# B&R Automation Studio project Stojan2
Automation Studio 4.0.18.71 SP

## Configuration Config1

CPU , AutomationRuntime P3.09, Build 4.1.2

### Task classes (Cpu.sw)
```

```

### Hardware
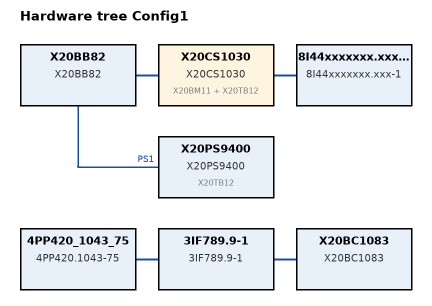
```
3IF789.9-1 : 3IF789.9-1 v1.1.3.0  [SS -> 4PP420_1043_75.SS1]
4PP420_1043_75 : 4PP420.1043-75 v1.0.0.0
  Cyclic1Duration = 10000
  Cyclic1Tolerance = 10000
  Cyclic2Duration = 20000
  Cyclic2Tolerance = 20000
  Cyclic3Duration = 50000
  Cyclic3Tolerance = 50000
  Cyclic4Duration = 100000
  Cyclic4Tolerance = 100000
  Cyclic5Duration = 200000
  Cyclic5Tolerance = 200000
  Cyclic6Duration = 500000
  Cyclic6Tolerance = 500000
  Cyclic7Duration = 1000000
  Cyclic7Tolerance = 1000000
  Cyclic8Duration = 10000
  Cyclic8Tolerance = 30000000
8I44xxxxxxx.xxx-1 : 8I44xxxxxxx.xxx-1 v1.1.3.0  [SER1 -> X20CS1030.IF1 (NodeNumber=10)]
  Supervision = off
  COD = 0
X20BB82 : X20BB82 v1.0.0.0
  Connector IF1:
    CycleTime = 1000
X20BC1083 : X20BC1083 v1.3.6.0  [PLK1 -> 3IF789.9-1.IF2 (NodeNumber=1); SL -> X20BB82.SL1]
X20BM11 : X20BM11 v1.0.0.0  [X2X1 -> X20BB82.IF1]
X20CS1030 : X20CS1030 v1.3.0.0  [SS1 -> X20TB12a.SS; SL -> X20BM11.SL1]
  Connector IF1:
    Baudrate = 19200
    DeviceType = RS485
    ActivateMODBUSRTU = 1
X20PS9400 : X20PS9400 v1.0.2.0  [SS1 -> X20TB12.SS; PS -> X20BB82.PS1]
X20TB12 : X20TB12 v1.0.0.0
X20TB12a : X20TB12 v1.0.0.0
```

## Logical view

Binary libraries used (declarations not repeated): operator, runtime, astime, AsIecCon, AsIOAcc


### Program Logical/ACPi (IEC)

#### ACPi.st - Cyclic code
```iecst
(********************************************************************
 * COPYRIGHT --
 ********************************************************************
 * Program: ACPi
 * File: ACPi.st
 * Author: vancurar
 * Created: 22.10.2012
 ********************************************************************
 * Implementation of program ACPi
 ********************************************************************)

PROGRAM _INIT
	LFRD_Output;

END_PROGRAM

PROGRAM _CYCLIC

	CASE ETAD_Input AND 16#FF  OF
		16#40, 16#50: (* Switch on disabled *)
		CMDD_Output := 16#0006;

		16#21, 16#31: (*Ready to switch on *)
		IF switchOn THEN
			CMDD_Output := 16#0007;
		END_IF

		16#33, 16#23: (*Switched on *)
		CMDD_Output := 16#000F;

		16#37, 16#27: (*Operation enabled *)
		IF NOT switchOn THEN
			CMDD_Output := 16#0006;
		END_IF

		IF quickStop THEN
			CMDD_Output := 16#0002;
		END_IF

		16#17, 16#07: (*Quick stop active *)
		quickStop := FALSE;
		switchOn := FALSE;
		CMDD_Output := 16#0000;
	END_CASE;

	IF (ETAD_Input AND 16#F) = 8 THEN (* Fault *)
		IF reset THEN
			reset := FALSE;
			CMDD_Output := 16#0080;
		END_IF
	END_IF

END_PROGRAM
```

#### ACPi.var - Local variables
```iecst
(********************************************************************
 * COPYRIGHT --
 ********************************************************************
 * Program: x64task
 * File: x64task.var
 * Author: vancurar
 * Created: November 15, 2011
 ********************************************************************
 * Local variables of program x64task
 ********************************************************************)
VAR
	CMDD_Output : UINT; (*control word*)
	ETAD_Input : UINT; (*status word*)
	switchOn : BOOL;
	LFRD_Output : INT; (*set speed [rpm]*)
	quickStop : BOOL;
	reset : BOOL;
END_VAR
```

### Program Logical/x64_rsc (IEC)

#### x64_rscCyclic.st - Cyclic code
```iecst
(********************************************************************
 * COPYRIGHT -- Bernecker + Rainer
 ********************************************************************
 * Program: x64_rsc
 * File: x64_rscCyclic.st
 * Author: vancurar
 * Created: September 15, 2014
 ********************************************************************
 * Implementation of program x64_rsc
 ********************************************************************)

PROGRAM _CYCLIC

	AsIOAccRead_0.enable := 1;
	AsIOAccRead_0.pDeviceName := ADR('SL1.SS1.IF1.ST1');
	AsIOAccRead_0.pChannelName := ADR('RSC_Input');
	AsIOAccRead_0();

END_PROGRAM
```

#### x64_rsc.var - Local variables
```iecst
(********************************************************************
 * COPYRIGHT -- Bernecker + Rainer
 ********************************************************************
 * Program: x64_rsc
 * File: x64_rsc.var
 * Author: vancurar
 * Created: September 15, 2014
 ********************************************************************
 * Local variables of program x64_rsc
 ********************************************************************)
VAR
	AsIOAccRead_0 : AsIOAccRead;
	ModuleOk : BOOL;
END_VAR
```
